{attribute addProperty BoxType "EL6201-0000-0017"}
{attribute addProperty Id "Slave_14A_DO0BIT10.125105Slave_14A_DO1BIT10.125106Slave_14A_DO2BIT10.125107Slave_14A_DO3BIT10.125108Slave_14B_DO0BIT10.125109Slave_14B_DO1BIT10.125110Slave_14B_DO2BIT10.125111Slave_14B_DO3BIT10.125112"}
{attribute addProperty CRC "1104667462"}
{attribute addProperty SizeInBites "8"}
{attribute addProperty SizeInBytes "1"}
TYPE Slave_14_Outputs_41D7E346 :
STRUCT
	{attribute addProperty Name "Slave_14A_DO0"}
	Slave_14A_DO0 : BIT;
	{attribute addProperty Name "Slave_14A_DO1"}
	Slave_14A_DO1 : BIT;
	{attribute addProperty Name "Slave_14A_DO2"}
	Slave_14A_DO2 : BIT;
	{attribute addProperty Name "Slave_14A_DO3"}
	Slave_14A_DO3 : BIT;
	{attribute addProperty Name "Slave_14B_DO0"}
	Slave_14B_DO0 : BIT;
	{attribute addProperty Name "Slave_14B_DO1"}
	Slave_14B_DO1 : BIT;
	{attribute addProperty Name "Slave_14B_DO2"}
	Slave_14B_DO2 : BIT;
	{attribute addProperty Name "Slave_14B_DO3"}
	Slave_14B_DO3 : BIT;
END_STRUCT
END_TYPE

(* stored: Version 1.2.0.0, ProductVersion 3.1.4024.9
   DUT Slave_14_Outputs_41D7E346: Id {27567024-9aea-47a9-bf87-47eba643f1b2} *)
